TYPE DUT_SENSOR_DATAS_8 :
UNION
	data_lreal:REAL;
	data_byte:ARRAY[0..3] OF BYTE;
END_UNION
END_TYPE

(* stored: Version 1.1.0.1, ProductVersion 3.1.4024.6
   DUT DUT_SENSOR_DATAS_8: Id {0151ac6e-d464-41e4-bf09-06b6f377a39d} *)
